TYPE T_UDP_INFO :
STRUCT
	bDriverInitialization: BOOL; // Indication of whether the realtime driver is properly initialized.  
	nReceivedPackets: UDINT; // counter the number of times the diagnostic data was sent.
	uSenderAddress: T_IP_ADDRESS;
	ipv4Adr : T_IPv4Addr := '';
	lrNotification: LREAL; // timestamp of the last sent
	sNotification: STRING;
END_STRUCT
END_TYPE

(* stored: Version 1.1.0.1, ProductVersion 3.1.4024.11
   DUT T_UDP_INFO: Id {c3edef04-eb42-4ac0-8bf0-136f7e8fdce9} *)
